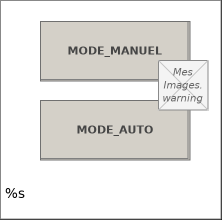
VISUALIZATION VISU_MODE_MARCHE  // 222x220
VAR_IN_OUT
	m_Input_MACHINE : BLOCK_MODE_MARCHE_V2_0;
END_VAR
    Rectangle (0,0 222x220)
    Rectangle (2,170 219x47), "%s", text list: 'TextList_STATE_Mode_Marche', text index: m_Input_MACHINE.STATUS
    Button (40,21 150x60), "MODE_MANUEL", colour toggle: m_Input_MACHINE.STATE_Manu, input disabled if: NOT m_Input_MACHINE.AUTOR_Manu_Ihm OR PRG_SEC.VERROU OR NOT PRG_USER.ACTU_USER.MAINTENANCE
        OnMouseClick: toggle m_Input_MACHINE.M_Manu
    Button (40,100 150x60), "MODE_AUTO", colour toggle: m_Input_MACHINE.STATE_Auto, input disabled if: NOT m_Input_MACHINE.AUTOR_Auto_Ihm
        OnMouseClick: toggle m_Input_MACHINE.M_Auto
    Image (158,60 50x50), invisible if: .STATE_Charg_Persistentes_Ok, image: MesImages.warning
END_VISUALIZATION

(* stored: Version 1.1.0.1, ProductVersion 3.1.4024.12
   Visu VISU_MODE_MARCHE: Id {3121ed37-0c0e-4838-9b0c-700c3c13e1b5} *)
